(*
	The function block serves as the basic implementation of an event listener.
	New messages and state changes of alarms can be recognized through the overwriting of the event-driven
	methods.
*)
FUNCTION_BLOCK FB_AlarmListener EXTENDS FB_ListenerBase2
VAR
(*POUs*)
	fbRequestEventText:			FB_RequestEventText;
(*Property vars*)
	udnLastEventID: 			UDINT;
	ulnLastEventTimeStamp: 		ULINT;
	sLastEventText: 			STRING;
	bReqEventText: 				BOOL;
	bAlarmRaised:				BOOL;
	bAlarmConfirmed:			BOOL;
	bAlarmCleared:				BOOL;
END_VAR

METHOD Execute : HRESULT
VAR_INPUT
END_VAR
Execute := SUPER^.Execute(); //retrieve events

//retrieve the text of a message
IF 	bReqEventText AND fbRequestEventText.bError THEN 
	sLastEventText := 'Error';
	bReqEventText := FALSE; 
ELSIF bReqEventText AND NOT  fbRequestEventText.bBusy THEN
	fbRequestEventText.GetString(sLastEventText, SIZEOF(sLastEventText));
	bReqEventText := FALSE;
END_IF
END_METHOD

METHOD OnAlarmCleared : HRESULT
VAR_INPUT
	fbEvent:	REFERENCE TO FB_TcEvent;
END_VAR
//Get alarm ID 
udnLastEventID := fbEvent.nEventId;
//Get alarm time stamp
ulnLastEventTimeStamp := fbEvent.nTimestamp;
//Send request to get alarm text 
fbRequestEventText.Request(eventClass := fbEvent.EventClass, nEventId := fbEvent.nEventId, nLangId := 1033, ipArgs := fbEvent.ipArguments);
bReqEventText := TRUE;
//Validate alarm cleared
bAlarmCleared := TRUE;
END_METHOD

METHOD OnAlarmConfirmed : HRESULT
VAR_INPUT
	fbEvent:	REFERENCE TO FB_TcEvent;
END_VAR
//Get alarm ID 
udnLastEventID := fbEvent.nEventId;
//Get alarm time stamp
ulnLastEventTimeStamp := fbEvent.nTimestamp;
//Send request to get alarm text 
fbRequestEventText.Request(eventClass := fbEvent.EventClass, nEventId := fbEvent.nEventId, nLangId := 1033, ipArgs := fbEvent.ipArguments);
bReqEventText := TRUE;
//Validate alarm confirmed
bAlarmConfirmed := TRUE;
END_METHOD

METHOD OnAlarmRaised : HRESULT
VAR_INPUT
	fbEvent:	REFERENCE TO FB_TcEvent;
END_VAR
//Get alarm ID 
udnLastEventID := fbEvent.nEventId;
//Get alarm time stamp
ulnLastEventTimeStamp := fbEvent.nTimestamp;
//Send request to get alarm text 
fbRequestEventText.Request(eventClass := fbEvent.EventClass, nEventId := fbEvent.nEventId, nLangId := 1033, ipArgs := fbEvent.ipArguments);
bReqEventText := TRUE;
//Validate alarm raised
bAlarmRaised := TRUE;
END_METHOD

PROPERTY pAlarmCleared : BOOL
GET
pAlarmCleared := bAlarmCleared;
END_GET
SET
bAlarmCleared := pAlarmCleared;
END_SET
END_PROPERTY

PROPERTY pAlarmConfirmed : BOOL
GET
pAlarmConfirmed := bAlarmConfirmed;
END_GET
SET
bAlarmConfirmed := pAlarmConfirmed;
END_SET
END_PROPERTY

PROPERTY pAlarmRaised : BOOL
GET
pAlarmRaised := bAlarmRaised;
END_GET
SET
bAlarmRaised := pAlarmRaised;
END_SET
END_PROPERTY

PROPERTY pLastEventID : udint
GET
pLastEventID := udnLastEventID;
END_GET
END_PROPERTY

PROPERTY pLastEventText : string
GET
pLastEventText := sLastEventText;
END_GET
END_PROPERTY

PROPERTY pLastEventTimeStamp : ulint
GET
pLastEventTimeStamp := ulnLastEventTimeStamp;
END_GET
END_PROPERTY

END_FUNCTION_BLOCK

(* stored: Version 1.1.0.1, ProductVersion 3.1.4024.12
   POU FB_AlarmListener: Id {f5a091c5-13de-4239-b65c-02c4e0e19b4c}, SpecialFunc None
   Method Execute: Id {0071f062-5957-43c3-9046-60c4e16f3ea4}
   Method OnAlarmCleared: Id {1ec6d741-b38b-4a00-8232-77d9e322dc0b}
   Method OnAlarmConfirmed: Id {fac9c096-a6a5-4998-bbbd-a22e87eccca0}
   Method OnAlarmRaised: Id {4d95c52d-1f22-46fb-ad4e-7340e87fbedc}
   Property pAlarmCleared: Id {1af81927-7f7e-406e-9560-8f90e695b1d5}
   Get Get: Id {06f9264c-c756-4aeb-9490-4385c62fab5a}
   Set Set: Id {b44a232f-f2d4-46ab-b544-205ffce1061b}
   Property pAlarmConfirmed: Id {869e3f20-0487-4e3f-b8cc-431dfb91ec06}
   Get Get: Id {c0d6ccf1-f7e7-4ee8-b94a-726946365537}
   Set Set: Id {e4e761e7-4645-456c-8743-e9ceb79744e3}
   Property pAlarmRaised: Id {2a1e2dc2-a3cc-4af8-9a1b-f0c80cece87e}
   Get Get: Id {780c5a83-f437-40b7-a93c-3e3420e31968}
   Set Set: Id {ef17bef6-a298-4230-ac4e-e8caa27be8c5}
   Property pLastEventID: Id {c29fac3b-38c2-469a-88f5-3e8c1750c274}
   Get Get: Id {aaa1dedf-1fb6-42df-bc0e-9516ced32b66}
   Property pLastEventText: Id {8fc69a74-daba-4841-af33-9ba221d35839}
   Get Get: Id {ffe48195-99b8-47c6-a8dd-9eeab89e9dec}
   Property pLastEventTimeStamp: Id {7b5fa08c-0604-4f4e-a9a5-e7023ad8a822}
   Get Get: Id {f7cab8d3-1964-4489-9587-8c83315a3875} *)
